(* IEC 61131-3 sources: com.logicals.lc3.examples/HttpPost/src, 1 file *)

(* ---- HttpPostExampleProgram.iecst ---- *)
PROGRAM HttpPostExampleProgram
	VAR
	  status : DINT;
	END_VAR

	HttpPost(URL := 'http://192.168.1.152:8000/', PostFields := 'name=daniel&project=curl', ReturnCode => status, ENO => ENO);
END_PROGRAM
